FUNCTION_BLOCK INTERNAL_VAR_FB (* Simple FB with one algorithm *)
  (* Standard: 61499-1 *)
  (* Version 1.1, 2025-08-19, steamdragon *)
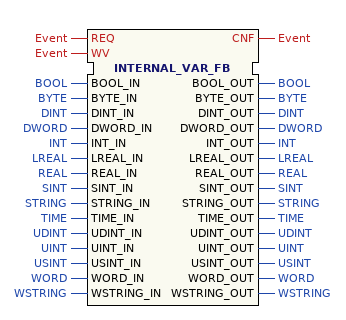
  EVENT_INPUT
    REQ; (* Normal Execution Request *)
    WV; (* Override internal Variables *)
  END_EVENT
  EVENT_OUTPUT
    CNF; (* Execution Confirmation *)
  END_EVENT
  VAR_INPUT
    BOOL_IN : BOOL; (* Manual Override *) {SET_ATTRIBUTE(VarConfig, true)}
    BYTE_IN : BYTE; {SET_ATTRIBUTE(VarConfig, true)}
    DINT_IN : DINT; {SET_ATTRIBUTE(VarConfig, true)}
    DWORD_IN : DWORD; {SET_ATTRIBUTE(VarConfig, true)}
    INT_IN : INT; {SET_ATTRIBUTE(VarConfig, true)}
    LREAL_IN : LREAL; {SET_ATTRIBUTE(VarConfig, true)}
    REAL_IN : REAL; {SET_ATTRIBUTE(VarConfig, true)}
    SINT_IN : SINT; {SET_ATTRIBUTE(VarConfig, true)}
    STRING_IN : STRING; {SET_ATTRIBUTE(VarConfig, true)}
    TIME_IN : TIME; {SET_ATTRIBUTE(VarConfig, true)}
    UDINT_IN : UDINT; {SET_ATTRIBUTE(VarConfig, true)}
    UINT_IN : UINT; {SET_ATTRIBUTE(VarConfig, true)}
    USINT_IN : USINT; {SET_ATTRIBUTE(VarConfig, true)}
    WORD_IN : WORD; {SET_ATTRIBUTE(VarConfig, true)}
    WSTRING_IN : WSTRING; {SET_ATTRIBUTE(VarConfig, true)}
  END_VAR
  VAR_OUTPUT
    BOOL_OUT : BOOL := FALSE; {SET_ATTRIBUTE(VarConfig, true)}
    BYTE_OUT : BYTE := 16#00; {SET_ATTRIBUTE(VarConfig, true)}
    DINT_OUT : DINT := 0; {SET_ATTRIBUTE(VarConfig, true)}
    DWORD_OUT : DWORD := 16#00000000; {SET_ATTRIBUTE(VarConfig, true)}
    INT_OUT : INT := 0; {SET_ATTRIBUTE(VarConfig, true)}
    LREAL_OUT : LREAL := 0.0; {SET_ATTRIBUTE(VarConfig, true)}
    REAL_OUT : REAL := 0.0; {SET_ATTRIBUTE(VarConfig, true)}
    SINT_OUT : SINT := 0; {SET_ATTRIBUTE(VarConfig, true)}
    STRING_OUT : STRING; {SET_ATTRIBUTE(VarConfig, true)}
    TIME_OUT : TIME := T#0ms; {SET_ATTRIBUTE(VarConfig, true)}
    UDINT_OUT : UDINT := 0; {SET_ATTRIBUTE(VarConfig, true)}
    UINT_OUT : UINT := 0; {SET_ATTRIBUTE(VarConfig, true)}
    USINT_OUT : USINT := 0; {SET_ATTRIBUTE(VarConfig, true)}
    WORD_OUT : WORD := 16#0000; {SET_ATTRIBUTE(VarConfig, true)}
    WSTRING_OUT : WSTRING; {SET_ATTRIBUTE(VarConfig, true)}
  END_VAR
END_FUNCTION_BLOCK
